(* CoDeSys 2.3.9.48 project: test.pro *)
(* Libraries: Standard.lib 8.11.10 12:37:48, SYSLIBCALLBACK.LIB 8.11.10 12:37:48, SerComm.lib 31.5.11 09:06:48, Serial_Interface_01.lib 22.4.13 12:50:14 *)

(* PLC configuration (modules and I/O channels)
K-Bus [K_Bus] node 0, in %IB0 out %QB0
Fieldbus variables [FB_VARS] node 1, in %IB0 out %QB0
Flag variables [FLAG_VARS] node 2, in %IB0 out %QB0
Modbus-Master [MB_MASTER] node 3, in %IB0 out %QB0
*)

(* Task configuration *)
TASK Serial3 (PRIORITY := 1, INTERVAL := T#200ms);
	COM3();
END_TASK

(* POU COM3, ST *)
PROGRAM COM3
VAR
	PT_SendStr : POINTER TO ARRAY[0..255] OF BYTE;
	PT_TmpStr : POINTER TO ARRAY[0..255] OF BYTE;
	SendString : STRING:='070';
	M_RECVSTR : BOOL:=FALSE;
	M_SENDSTR : BOOL:=TRUE;
(* Communicationparams FOR 750-65x/003-000 only*)
	wBaudRate : WORD := 5760;
	bDataBits : BYTE := 8;
	bParity : BYTE := 0; (*0=NO*)
	bFlowControl : BYTE := 4; (*1=XON/XOFF*)
	i : INT;
	in_COM_Port : INT := INT#3;
(*COM *******)
	COM : SERIAL_INTERFACE;
	xOpenPort : BOOL := TRUE;
	xInitPort : BOOL;
	xSendActive : BOOL;
	ReceiveBuffer: typRing_Buffer;
	ReceiveBufferOldIndex : INT;
	ReceiveString : STRING(255);
	pReceiveStr : POINTER TO ARRAY[0..255] OF BYTE;
	bERROR : BYTE :=16#00;
	Messwert01: REAL;
END_VAR
COM( bCOM_PORT_NR := INT_TO_BYTE(in_COM_Port),
  cbBAUDRATE        := wBaudRate,
  cbsBYTESIZE       := bDataBits,
  cpPARITY          := bParity,
  csSTOPBITS        := STOPBITS_1,
  cfFLOW_CONTROL    := bFlowControl,
  utRECEIVE_BUFFER  := ReceiveBuffer,
  ptSEND_BUFFER     := ADR(SendString),
  xINIT             := xInitPort,
  xOPEN_COM_PORT    := xOpenPort,
  iBYTES_TO_SEND    := LEN(SendString)+1,
  xSTART_SEND       := M_SENDSTR);
bERROR:=COM.bERROR;

IF pReceiveStr = 0 THEN (*Empfangspuffer mit Adresse von Empfangsstring initialisieren*)

  pReceiveStr := ADR( ReceiveString );

END_IF;

IF ReceiveBuffer.Index>0 THEN (*Neue Daten empfangen*)

IF ReceiveBuffer.Data[ ReceiveBuffer.Index-1 ] = 16#0A THEN (*16#0A=LF(Linefeed)*)

     FOR i:=0 TO 255 DO

        pReceiveStr^[i]:=16#00;  (*Empfangspuffer löschen*)

     END_FOR;

     FOR i:=0 TO ReceiveBuffer.Index-1 DO

        pReceiveStr^[i] :=  ReceiveBuffer.Data[ i ]; (*Ringpufferdaten in Empfangspuffer kopieren*)

     END_FOR;

     M_RECVSTR:=TRUE;

     ReceiveBuffer.Index:=0; (*Index des Ringpuffers zurücksetzen*)

END_IF;

END_IF;

(*Messwert01 := (WORD_TO_REAL(WPACK(ReceiveBuffer.Data[0], ReceiveBuffer.Data[1])));*)
END_PROGRAM

(* POU PLC_PRG, ST *)
PROGRAM PLC_PRG
VAR
	PT_SendStr : POINTER TO ARRAY[0..255] OF BYTE;
	PT_TmpStr : POINTER TO ARRAY[0..255] OF BYTE;
	SendString : STRING:='070';
	M_RECVSTR : BOOL:=FALSE;
	M_SENDSTR : BOOL:=TRUE;
(* Communicationparams FOR 750-65x/003-000 only*)
	wBaudRate : WORD := 5760;
	bDataBits : BYTE := 8;
	bParity : BYTE := 0; (*0=NO*)
	bFlowControl : BYTE := 4; (*1=XON/XOFF*)
	i : INT;
	in_COM_Port : INT := INT#2;
(*COM *******)
	COM : SERIAL_INTERFACE;
	xOpenPort : BOOL := TRUE;
	xInitPort : BOOL;
	xSendActive : BOOL;
	ReceiveBuffer: typRing_Buffer;
	ReceiveBufferOldIndex : INT;
	ReceiveString : STRING(255);
	pReceiveStr : POINTER TO ARRAY[0..255] OF BYTE;
	bERROR : BYTE :=16#00;
	Messwert01: REAL;
END_VAR
COM( bCOM_PORT_NR := INT_TO_BYTE(in_COM_Port),
  cbBAUDRATE        := wBaudRate,
  cbsBYTESIZE       := bDataBits,
  cpPARITY          := bParity,
  csSTOPBITS        := STOPBITS_1,
  cfFLOW_CONTROL    := bFlowControl,
  utRECEIVE_BUFFER  := ReceiveBuffer,
  ptSEND_BUFFER     := ADR(SendString),
  xINIT             := xInitPort,
  xOPEN_COM_PORT    := xOpenPort,
  iBYTES_TO_SEND    := LEN(SendString)+1,
  xSTART_SEND       := M_SENDSTR);
bERROR:=COM.bERROR;

IF pReceiveStr = 0 THEN (*Empfangspuffer mit Adresse von Empfangsstring initialisieren*)

  pReceiveStr := ADR( ReceiveString );

END_IF;

IF ReceiveBuffer.Index>0 THEN (*Neue Daten empfangen*)

IF ReceiveBuffer.Data[ ReceiveBuffer.Index-1 ] = 16#0A THEN (*16#0A=LF(Linefeed)*)

     FOR i:=0 TO 255 DO

        pReceiveStr^[i]:=16#00;  (*Empfangspuffer löschen*)

     END_FOR;

     FOR i:=0 TO ReceiveBuffer.Index-1 DO

        pReceiveStr^[i] :=  ReceiveBuffer.Data[ i ]; (*Ringpufferdaten in Empfangspuffer kopieren*)

     END_FOR;

     M_RECVSTR:=TRUE;

     ReceiveBuffer.Index:=0; (*Index des Ringpuffers zurücksetzen*)

END_IF;

END_IF;

(*Messwert01 := (WORD_TO_REAL(WPACK(ReceiveBuffer.Data[0], ReceiveBuffer.Data[1])));*)
END_PROGRAM
